FUNCTION_BLOCK FB_MotionBPTM_Test EXTENDS TcUnit.FB_TestSuite
(*
    Test the functionality of the motion bptm,
    Which is just a bptm wrapped up with a set of n motors.
    We're basically just making sure that we push the done button at the appropriate time.
    Direct tests of BPTM itself are reserved for the pmps library.

    The BPTM takes care of these executions across multiple cycles,
    so these tests must implement timeouts.
*)
VAR
    astMotionStage: ARRAY[1..MotionConstants.MAX_STATE_MOTORS] OF ST_MotionStage;
    stGoal1: ST_DbStateParams;
    stGoal2: ST_DbStateParams;
    stTrans: ST_DbStateParams;
    stNoBeam: ST_BeamParams;
END_VAR


stGoal1.stBeamParams := PMPS_GVL.cstFullBeam;
stGoal1.nRequestAssertionID := 1;
stGoal1.sPmpsState := 'stGoal1';
stGoal2.stBeamParams := PMPS_GVL.cstFullBeam;
stGoal2.stBeamParams.nTran := 0.5;
stGoal2.nRequestAssertionID := 2;
stGoal2.sPmpsState := 'stGoal2';
stTrans.stBeamParams := PMPS_GVL.cst0RateBeam;
stTrans.nRequestAssertionID := 3;
stTrans.sPmpsState := 'stTrans';

// Just put a blanket global no beam so these won't wait for any changes ever
PMPS_GVL.stCurrentBeamParameters := stNoBeam;
TestInit();
Test3dMove();
TestNoMove();
TestCount();


METHOD AssertInPool
VAR_IN_OUT
    fbArbiter: FB_Arbiter;
    stDbStateParams: ST_DbStateParams;
END_VAR
VAR_INPUT
    bInPool: BOOL;
    sContext: STRING;
END_VAR

IF bInPool THEN
    AssertTrue(
        fbArbiter.CheckRequestInPool(stDbStateParams.nRequestAssertionID),
        CONCAT(CONCAT(stDbStateParams.sPmpsState, ' Beam parameters were not in the pool '), sContext),
    );
ELSE
    AssertFalse(
        fbArbiter.CheckRequestInPool(stDbStateParams.nRequestAssertionID),
        CONCAT(CONCAT(stDbStateParams.sPmpsState, ' Beam parameters unexpectedly found in the pool '), sContext),
    );
END_IF
END_METHOD


METHOD SetMotorDone
VAR_INPUT
END_VAR

// Force post-move state
astMotionStage[1].bBusy := FALSE;
astMotionStage[1].bDone := TRUE;
astMotionStage[2].bBusy := FALSE;
astMotionStage[2].bDone := TRUE;
astMotionStage[3].bBusy := FALSE;
astMotionStage[3].bDone := TRUE;
END_METHOD


METHOD SetMotorMoving
VAR_INPUT
END_VAR

// Force a moving but not done state
astMotionStage[1].bBusy := TRUE;
astMotionStage[1].bDone := FALSE;
astMotionStage[2].bBusy := TRUE;
astMotionStage[2].bDone := FALSE;
astMotionStage[3].bBusy := TRUE;
astMotionStage[3].bDone := FALSE;
END_METHOD


METHOD SetMotorStartup
VAR_INPUT
END_VAR

// Force some sort of default looking state
astMotionStage[1].bBusy := FALSE;
astMotionStage[1].bDone := FALSE;
astMotionStage[2].bBusy := FALSE;
astMotionStage[2].bDone := FALSE;
astMotionStage[3].bBusy := FALSE;
astMotionStage[3].bDone := FALSE;
END_METHOD


METHOD Test3dMove : BOOL
(*
    Can we safely do a 3d move?
*)
VAR_INST
    fbBptm: FB_MotionBPTM;
    fbArbiter: FB_Arbiter(2);
    fbFFHWO: FB_HardwareFFOutput := (bAutoReset := TRUE);
    fbSubSysIO : FB_DummyArbIO;

    nState: UINT;
    tonTimer: TON;
END_VAR

TEST('Test3DMove');

tonTimer(
    IN:=TRUE,
    PT:=T#5s,
);
IF tonTimer.Q THEN
    nState := 4;
END_IF

CASE nState OF
    0:
        // Establish baseline at Goal1
        SetMotorStartup();
        fbBptm(
            astMotionStage:=astMotionStage,
            fbArbiter:=fbArbiter,
            fbFFHWO:=fbFFHWO,
            stGoalParams:=stGoal1,
            stTransParams:=stTrans,
            nActiveMotorCount:=3,
            bEnable:=TRUE,
            bAtState:=TRUE,
        );
        IF fbBptm.bDone THEN
            nState := 1;
        END_IF
    1:
        // Request a move
        SetMotorStartup();
        fbBptm(
            astMotionStage:=astMotionStage,
            fbArbiter:=fbArbiter,
            fbFFHWO:=fbFFHWO,
            stGoalParams:=stGoal2,
            stTransParams:=stTrans,
            nActiveMotorCount:=3,
            bEnable:=TRUE,
            bAtState:=FALSE,
        );
        IF fbBptm.bTransitionAuthorized THEN
            // We should have transition and goal 2 asserts in
            AssertInPool(fbArbiter, stGoal1, FALSE, 'with trans auth');
            AssertInPool(fbArbiter, stGoal2, TRUE, 'with trans auth');
            AssertInPool(fbArbiter, stTrans, TRUE, 'with trans auth');
            nState := 2;
        END_IF
    2:
        // Simulate a move
        SetMotorMoving();
        fbBptm(
            astMotionStage:=astMotionStage,
            fbArbiter:=fbArbiter,
            fbFFHWO:=fbFFHWO,
            stGoalParams:=stGoal2,
            stTransParams:=stTrans,
            nActiveMotorCount:=3,
            bEnable:=TRUE,
            bAtState:=FALSE,
        );
        // Same situation as before
        AssertInPool(fbArbiter, stGoal1, FALSE, 'after move started');
        AssertInPool(fbArbiter, stGoal2, TRUE, 'after move started');
        AssertInPool(fbArbiter, stTrans, TRUE, 'after move started');
        nState := 3;
    3:
        // Move is done
        SetMotorDone();
        fbBptm(
            astMotionStage:=astMotionStage,
            fbArbiter:=fbArbiter,
            fbFFHWO:=fbFFHWO,
            stGoalParams:=stGoal2,
            stTransParams:=stTrans,
            nActiveMotorCount:=3,
            bEnable:=TRUE,
            bAtState:=TRUE,
        );
        IF fbBptm.bDone THEN
            // Dropped the transition assert
            AssertInPool(fbArbiter, stGoal1, FALSE, 'with move complete');
            AssertInPool(fbArbiter, stGoal2, TRUE, 'with move complete');
            AssertInPool(fbArbiter, stTrans, FALSE, 'with move complete');
            nState := 4;
        END_IF
    4:
        AssertFalse(
            tonTimer.Q,
            'Timeout in test',
        );
        TEST_FINISHED();
END_CASE

fbSubSysIO(
    LA:=fbArbiter,
    FFO:=fbFFHWO,
);
END_METHOD


METHOD TestCount
(*
    FB Should just error out if we forgot to give a count
*)
VAR_INST
    fbBptm: FB_MotionBPTM;
    fbArbiter: FB_Arbiter(1);
    fbFFHWO: FB_HardwareFFOutput := (bAutoReset := TRUE);

    tonWait: TON;
END_VAR

TEST('TestCount');

SetMotorStartup();
fbBptm(
    astMotionStage:=astMotionStage,
    fbArbiter:=fbArbiter,
    fbFFHWO:=fbFFHWO,
    stGoalParams:=stGoal1,
    stTransParams:=stTrans,
    bEnable:=True,
    bAtState:=True,
);
AssertTrue(
    fbBptm.bMotorCountError,
    'Did not properly error on missing motor count',
);

tonWait(
    IN:=TRUE,
    PT:=T#1s,
);
IF tonWait.Q THEN
    // Should have no arbiter activity at all
    AssertInPool(fbArbiter, stGoal1, FALSE, 'with bad count');
    AssertInPool(fbArbiter, stGoal2, FALSE, 'with bad count');
    AssertInPool(fbArbiter, stTrans, FALSE, 'with bad count');

    TEST_FINISHED();
END_IF
END_METHOD


METHOD TestInit : BOOL
(*
    If we initialize with still motors, do we get an arbiter request at the current goal? Hopefully we do.
*)
VAR_INST
    fbBptm: FB_MotionBPTM;
    fbArbiter: FB_Arbiter(1);
    fbFFHWO: FB_HardwareFFOutput := (bAutoReset := TRUE);
    fbSubSysIO : FB_DummyArbIO;

    tonTimer: TON;
END_VAR

TEST('TestInit');

SetMotorStartup();
fbBptm(
    astMotionStage:=astMotionStage,
    fbArbiter:=fbArbiter,
    fbFFHWO:=fbFFHWO,
    stGoalParams:=stGoal1,
    stTransParams:=stTrans,
    nActiveMotorCount:=3,
    bEnable:=True,
    bAtState:=True,
);
fbSubSysIO(
    LA:=fbArbiter,
    FFO:=fbFFHWO,
);

tonTimer(
    IN:=TRUE,
    PT:=T#5s,
);
IF tonTimer.Q OR fbBptm.bDone THEN
    AssertFalse(
        tonTimer.Q,
        'Timeout in test',
    );
    // We should have a request in the pool for goal 1 but not for transition
    // If no request are in the pool, we may come up in a no protection state!
    // If both requests are in the pool, we may come up in a too much blocking beam state!
    AssertInPool(fbArbiter, stGoal1, TRUE, 'at startup');
    AssertInPool(fbArbiter, stTrans, FALSE, 'at startup');

    TEST_FINISHED();
END_IF
END_METHOD


METHOD TestNoMove
(*
    In place transitions should work at startup and also at done positions.
*)
VAR_INST
    fbBptm: FB_MotionBPTM;
    fbArbiter: FB_Arbiter(1);
    fbFFHWO: FB_HardwareFFOutput := (bAutoReset := TRUE);
    fbSubSysIO : FB_DummyArbIO;

    nState: UINT;
    tonTimer: TON;
END_VAR

TEST('TestNoMove');

tonTimer(
    IN:=TRUE,
    PT:=T#5s,
);
IF tonTimer.Q THEN
    nState := 3;
END_IF

CASE nState OF
    0:
        SetMotorStartup();
        fbBptm(
            astMotionStage:=astMotionStage,
            fbArbiter:=fbArbiter,
            fbFFHWO:=fbFFHWO,
            stGoalParams:=stGoal1,
            stTransParams:=stTrans,
            nActiveMotorCount:=3,
            bEnable:=True,
            bAtState:=True,
        );
        IF fbBptm.bDone THEN
            nState := 1;
        END_IF
    1:
        SetMotorStartup();
        // NOTE: we kept bAtState TRUE the whole time, so this should be a completed in-place transition
        fbBptm(
            astMotionStage:=astMotionStage,
            fbArbiter:=fbArbiter,
            fbFFHWO:=fbFFHWO,
            stGoalParams:=stGoal2,
            stTransParams:=stTrans,
            nActiveMotorCount:=3,
            bEnable:=True,
            bAtState:=True,
        );
        IF fbBptm.bDone THEN
            // Only Goal2 should be in the pool
            AssertInPool(fbArbiter, stGoal1, FALSE, 'after switching goals (1)');
            AssertInPool(fbArbiter, stGoal2, TRUE, 'after switching goals (1)');
            AssertInPool(fbArbiter, stTrans, FALSE, 'after switching goals (1)');
            nState := 2;
        END_IF
    2:
        // Repeat from a done position!
        SetMotorDone();
        fbBptm(
            astMotionStage:=astMotionStage,
            fbArbiter:=fbArbiter,
            fbFFHWO:=fbFFHWO,
            stGoalParams:=stGoal1,
            stTransParams:=stTrans,
            nActiveMotorCount:=3,
            bEnable:=True,
            bAtState:=True,
        );
        IF fbBptm.bDone THEN
            // Only Goal1 should be in the pool
            AssertInPool(fbArbiter, stGoal1, TRUE, 'after switching goals (2)');
            AssertInPool(fbArbiter, stGoal2, FALSE, 'after switching goals (2)');
            AssertInPool(fbArbiter, stTrans, FALSE, 'after switching goals (2)');
            nState := 3;
        END_IF
    3:
        AssertFalse(
            tonTimer.Q,
            'Timeout in test',
        );
        TEST_FINISHED();
END_CASE

fbSubSysIO(
    LA:=fbArbiter,
    FFO:=fbFFHWO,
);
END_METHOD

END_FUNCTION_BLOCK

(* stored: Version 1.1.0.1
   POU FB_MotionBPTM_Test: Id {74dc5407-5bbf-4092-b438-4ab304d6e18f}, SpecialFunc None
   Method AssertInPool: Id {5d2e8161-724f-4980-ba8a-e3e41656d95f}
   Method SetMotorDone: Id {387bbfef-8396-472d-9e1b-a94d57b4b859}
   Method SetMotorMoving: Id {9274df44-2fe4-4272-82fa-4af8d13cf00c}
   Method SetMotorStartup: Id {23decd21-83c3-4f7e-bc90-32e7f7f554e3}
   Method Test3dMove: Id {9921e26f-7be4-494e-96b8-8a52185f8503}
   Method TestCount: Id {210e6655-146a-47df-9045-4ed85f85c10f}
   Method TestInit: Id {aa2dec78-fff0-42b9-a0fa-1c26187b6d46}
   Method TestNoMove: Id {fb9625b7-e60b-4c6d-b5c7-290ec4718085} *)
